FUNCTION_BLOCK FB_List_Test EXTENDS TcUnit.FB_TestSuite
VAR
END_VAR

THIS^.Size_And_Is_Empty();
THIS^.Append_And_Get();
THIS^.Prepend_And_Get();
THIS^.Append_And_Reverse();
THIS^.Append_Find_And_Get();
THIS^.Remove_Tests();
THIS^.Set_And_Get();

// Test appending multiple elements and verify their order and values using the get method.
METHOD Append_And_Get
VAR_INST
	fbList 		: FB_List;
	
	arbValue 	: ARRAY[0..2] OF BOOL := [TRUE, TRUE];
	arnValue 	: ARRAY[0..2] OF INT := [33, 33];
	arsValue 	: ARRAY[0..2] OF STRING := ['I love cats.', 'I love cats.'];
	arwsValue 	: ARRAY[0..2] OF WSTRING := ["I love dogs.", "I love dogs."];
	arfValue 	: ARRAY[0..2] OF LREAL := [21.3, 21.3];
END_VAR
TcUnit.TEST('Append_And_Get');

	fbList
		.Append(arbValue[0])
		.Append(arnValue[0])
		.Append(arsValue[0])
		.Append(arwsValue[0])
		.Append(arfValue[0]);
		
	fbList
		.Get(0, arbValue[2])
		.Get(1, arnValue[2])
		.Get(2, arsValue[2])
		.Get(3, arwsValue[2])
		.Get(4, arfValue[2]);
		
	THIS^.AssertEquals_DINT(5, fbList._Count, 'List item count must be 5 after after appending items to list.');
	THIS^.AssertEquals_BOOL(arbValue[1], arbValue[2], 'Appended BOOL item is not what is expected after the get operation.');
	THIS^.AssertEquals_INT(arnValue[1], arnValue[2], 'Appended INT item is not what is expected after the get operation.');
	THIS^.AssertEquals_STRING(arsValue[1], arsValue[2], 'Appended STRING item is not what is expected after the get operation.');
	THIS^.AssertEquals_WSTRING(arwsValue[1], arwsValue[2], 'Appended STRING item is not what is expected after the get operation.');
	THIS^.AssertEquals_LREAL(arfValue[1], arfValue[2],0.01, 'Appended LREAL item is not what is expected after the get operation.');

	TEST_FINISHED();
END_METHOD

// Test appending multiple elements, reversing their order and verifiying their order and values using the get method.
METHOD Append_And_Reverse
VAR_INST
	fbList 		: FB_List;
	
	arbValue 	: ARRAY[0..2] OF BOOL := [TRUE, TRUE];
	arnValue 	: ARRAY[0..2] OF INT := [33, 33];
	arsValue 	: ARRAY[0..2] OF STRING := ['I love cats.', 'I love cats.'];
	arwsValue 	: ARRAY[0..2] OF WSTRING := ["I love dogs.", "I love dogs."];
	arfValue 	: ARRAY[0..2] OF LREAL := [21.3, 21.3];
END_VAR
TcUnit.TEST('Append_And_Reverse');

	fbList
		.Append(arbValue[0])
		.Append(arnValue[0])
		.Append(arsValue[0])
		.Append(arwsValue[0])
		.Append(arfValue[0])
		.Reverse();
		
	fbList
		.Get(4, arbValue[2])
		.Get(3, arnValue[2])
		.Get(2, arsValue[2])
		.Get(1, arwsValue[2])
		.Get(0, arfValue[2]);
		
	THIS^.AssertEquals_DINT(5, fbList._Count, 'List item count must be 5 after after appending items to list.');
	THIS^.AssertEquals_BOOL(arbValue[1], arbValue[2], 'Appended BOOL item is not what is expected after the get operation.');
	THIS^.AssertEquals_INT(arnValue[1], arnValue[2], 'Appended INT item is not what is expected after the get operation.');
	THIS^.AssertEquals_STRING(arsValue[1], arsValue[2], 'Appended STRING item is not what is expected after the get operation.');
	THIS^.AssertEquals_WSTRING(arwsValue[1], arwsValue[2], 'Appended STRING item is not what is expected after the get operation.');
	THIS^.AssertEquals_LREAL(arfValue[1], arfValue[2],0.01, 'Appended LREAL item is not what is expected after the get operation.');

	TEST_FINISHED();
END_METHOD

// Test appending multiple elements, finds them and verify values using the get method.
METHOD Append_Find_And_Get
VAR_INST
	fbList 		: FB_List;
	Idx 		: ARRAY[0..4] OF T_Position;
	arbValue 	: ARRAY[0..2] OF BOOL := [TRUE, TRUE];
	arnValue 	: ARRAY[0..2] OF INT := [33, 33];
	arsValue 	: ARRAY[0..2] OF STRING := ['I love cats.', 'I love cats.'];
	arwsValue 	: ARRAY[0..2] OF WSTRING := ["I love dogs.", "I love dogs."];
	arfValue 	: ARRAY[0..2] OF LREAL := [21.3, 21.3];
END_VAR
TcUnit.TEST('Append_Find_And_Get');

	fbList
		.Append(arbValue[0])
		.Append(arnValue[0])
		.Append(arsValue[0])
		.Append(arwsValue[0])
		.Append(arfValue[0]);

	// Make the strings dirty. 	
	arsValue[0] 	:= 'kjhsadkfjvhbkjhdfbkvsjhbfkvjhsbkfv';
	arwsValue[0] 	:= "kjhsadkfjvhbkjhdfbkvsjhbfkvjhsbkfv";
	arsValue[0] 	:= 'I love cats.';
	arwsValue[0] 	:= "I love dogs.";
		
	fbList
		.Search(arbValue[0], Index => Idx[0])
		.Search(arnValue[0], Index => Idx[1])
		.Search(arsValue[0], Index => Idx[2])
		.Search(arwsValue[0],Index => Idx[3])
		.Search(arfValue[0], Index => Idx[4]);
		
	fbList
		.Get(Idx[0], arbValue[2])
		.Get(Idx[1], arnValue[2])
		.Get(Idx[2], arsValue[2])
		.Get(Idx[3], arwsValue[2])
		.Get(Idx[4], arfValue[2]);
		
	THIS^.AssertEquals_DINT(5, fbList._Count, 'List item count must be 5 after after appending items to list.');
	THIS^.AssertEquals_BOOL(arbValue[1], arbValue[2], 'Appended BOOL item is not what is expected after the get operation.');
	THIS^.AssertEquals_INT(arnValue[1], arnValue[2], 'Appended INT item is not what is expected after the get operation.');
	THIS^.AssertEquals_STRING(arsValue[1], arsValue[2], 'Appended STRING item is not what is expected after the get operation.');
	THIS^.AssertEquals_WSTRING(arwsValue[1], arwsValue[2], 'Appended STRING item is not what is expected after the get operation.');
	THIS^.AssertEquals_LREAL(arfValue[1], arfValue[2],0.01, 'Appended LREAL item is not what is expected after the get operation.');

	TEST_FINISHED();
END_METHOD

// Test prepending multiple elements and verify their order and values using the get method.
METHOD Prepend_And_Get
VAR_INST
	fbList 		: FB_List;
	arsPrint 	: ARRAY[0..4] OF STRING;
	arbValue 	: ARRAY[0..2] OF BOOL := [TRUE, TRUE];
	arnValue 	: ARRAY[0..2] OF INT := [33, 33];
	arsValue 	: ARRAY[0..2] OF STRING := ['I love cats.', 'I love cats.'];
	arwsValue 	: ARRAY[0..2] OF WSTRING := ["I love dogs.", "I love dogs."];
	arfValue 	: ARRAY[0..2] OF LREAL := [21.3, 21.3];
END_VAR
TcUnit.TEST('Prepend_And_Get');

	fbList
		.Prepend(arbValue[0])
		.Prepend(arnValue[0])
		.Prepend(arsValue[0])
		.Prepend(arwsValue[0])
		.Prepend(arfValue[0]);
		
	fbList
		.Get(4, arbValue[2])
		.Get(3, arnValue[2])
		.Get(2, arsValue[2])
		.Get(1, arwsValue[2])
		.Get(0, arfValue[2]);
		
	THIS^.AssertEquals_DINT(5, fbList._Count, 'List item count must be 5 after after appending items to list.');
	THIS^.AssertEquals_BOOL(arbValue[1], arbValue[2], 'Appended BOOL item is not what is expected after the get operation.');
	THIS^.AssertEquals_INT(arnValue[1], arnValue[2], 'Appended INT item is not what is expected after the get operation.');
	THIS^.AssertEquals_STRING(arsValue[1], arsValue[2], 'Appended STRING item is not what is expected after the get operation.');
	THIS^.AssertEquals_WSTRING(arwsValue[1], arwsValue[2], 'Appended STRING item is not what is expected after the get operation.');
	THIS^.AssertEquals_LREAL(arfValue[1], arfValue[2],0.01, 'Appended LREAL item is not what is expected after the get operation.');

	TEST_FINISHED();
END_METHOD

// Test appending multiple elements, removing first item, verifying the size and values.
METHOD Remove_Tests
VAR_INST
	fbList 		: FB_List;
	i 			: T_Position;
	n 			: T_Capacity;
	arbValue 	: ARRAY[0..2] OF BOOL := [TRUE, TRUE];
	arnValue 	: ARRAY[0..2] OF INT := [33, 33];
	arsValue 	: ARRAY[0..2] OF STRING := ['I love cats.', 'I love cats.'];
	arwsValue 	: ARRAY[0..2] OF WSTRING := ["I love dogs.", "I love dogs."];
	arfValue 	: ARRAY[0..2] OF LREAL := [21.3, 21.3];
END_VAR
TcUnit.TEST('Remove_Tests');

	fbList
		.Append(arbValue[0])
		.Append(arnValue[0])
		.Append(arsValue[0])
		.Append(arwsValue[0])
		.Append(arfValue[0]);
		
	fbList
		.Remove(arbValue[0])
		.Get(0, arnValue[2]);
		
	THIS^.AssertEquals_DINT(4, fbList._Count, 'List item count must be 4 after appending and removing fisrt item at from the list.');
	THIS^.AssertEquals_INT(arnValue[1], arnValue[2],'');
	
	fbList
		.Prepend(arbValue[0])
		.Remove_At(2)
		.Get(2, arwsValue[2]);
		
	THIS^.AssertEquals_DINT(4, fbList._Count, 'List item count must be 4 after prepending removed item and removing item in index 2 of the list.');
	THIS^.AssertEquals_WSTRING(arwsValue[1], arwsValue[2], '');
	
	fbList
		.Insert(2, arsValue[0])
		.Remove_At(fbList._Count - 1)
		.Get(3, arwsValue[2]);
		
	THIS^.AssertEquals_DINT(4, fbList._Count, 'List item count must be 4 after inserting removed from index 2 item and removing the last item in the list.');
	THIS^.AssertEquals_WSTRING(arwsValue[1], arwsValue[2], '');

	n := fbList._Count;
	FOR i := 0 TO n DO
		fbList.Remove_At(fbList._Count - 1);
		END_FOR
		
	THIS^.AssertEquals_DINT(0, fbList._Count, 'List item count must be zero after removing all items from the back.');
	THIS^.AssertEquals_BOOL(TRUE, fbList._Is_Empty, 'List Is_Empty property must be zero TRUE removing all items from the back.');

	FOR i := 0 TO 4 DO fbList.Prepend(arwsValue); END_FOR
	
	THIS^.AssertEquals_DINT(5, fbList._Count, 'Failed to prepend items to list for checking removing all items from the front.');
	
	n := fbList._Count;
	FOR i := 0 TO n - 1 DO
		fbList.Remove_At(0);
		END_FOR
		
	THIS^.AssertEquals_DINT(0, fbList._Count, 'List item count must be zero after removing all items from the front.');
	THIS^.AssertEquals_BOOL(TRUE, fbList._Is_Empty, 'List Is_Empty property must be zero TRUE removing all items from the front.');

	TEST_FINISHED();
END_METHOD

// Test appending multiple elements and verify their order and values using the get method.
METHOD Set_And_Get
VAR_INST
	fbList 		: FB_List;
	
	arbValue 	: ARRAY[0..2] OF BOOL := [TRUE, TRUE];
	arnValue 	: ARRAY[0..2] OF INT := [33, 33];
	arsValue 	: ARRAY[0..2] OF STRING := ['I love cats.', 'I love cats.'];
	arwsValue 	: ARRAY[0..2] OF WSTRING := ["I love dogs.", "I love dogs."];
	arfValue 	: ARRAY[0..2] OF LREAL := [21.3, 21.3];
END_VAR
TcUnit.TEST('Set_And_Get');

	fbList
		.Resize(5)
		.Set(0, arbValue[0])
		.Set(1, arnValue[0])
		.Set(2, arsValue[0])
		.Set(3, arwsValue[0])
		.Set(4, arfValue[0]);
		
	fbList
		.Get(0, arbValue[2])
		.Get(1, arnValue[2])
		.Get(2, arsValue[2])
		.Get(3, arwsValue[2])
		.Get(4, arfValue[2]);
		
	THIS^.AssertEquals_DINT(5, fbList._Count, 'List item count must be 5 after after appending items to list.');
	THIS^.AssertEquals_BOOL(arbValue[1], arbValue[2], 'Get BOOL item is not what is expected after the get operation.');
	THIS^.AssertEquals_INT(arnValue[1], arnValue[2], 'Get INT item is not what is expected after the get operation.');
	THIS^.AssertEquals_STRING(arsValue[1], arsValue[2], 'Get STRING item is not what is expected after the get operation.');
	THIS^.AssertEquals_WSTRING(arwsValue[1], arwsValue[2], 'Get STRING item is not what is expected after the get operation.');
	THIS^.AssertEquals_LREAL(arfValue[1], arfValue[2],0.01, 'Get LREAL item is not what is expected after the get operation.');

	TEST_FINISHED();
END_METHOD

// 1) Test that a newly created FB_Array_List has an item count of 0 and is empty.
// 2) Test that after appending elements, the size increases accordingly and is no longer empty.
// 3) Test that after removing all elements, the size becomes 0 again and the list is empty.
METHOD Size_And_Is_Empty
VAR_INST
	fbList : FB_List;
	nValue : INT := 33;
	sValue : STRING := 'I love cats.';
END_VAR
TcUnit.TEST('Size_And_Is_Empty');

	THIS^.AssertEquals_DINT(0, fbList._Count, 'List item count must be 0.');
	THIS^.AssertEquals_BOOL(TRUE, fbList._Is_Empty, 'Is_Empty property didnt return TRUE.');
	
	fbList
		.Append(nValue)
		.Append(sValue);
	
	THIS^.AssertEquals_DINT(2, fbList._Count, 'List item count must be 2 after appending values.');
	THIS^.AssertEquals_BOOL(FALSE, fbList._Is_Empty, 'Is_Empty property didnt return FALSE after appending value.');
	
	fbList.Clear();
	
	THIS^.AssertEquals_DINT(0, fbList._Count, 'List item count must be 0 after clearing list.');
	THIS^.AssertEquals_BOOL(TRUE, fbList._Is_Empty, 'Is_Empty property didnt return TRUE after clearing list.');
	
	TEST_FINISHED();
END_METHOD

END_FUNCTION_BLOCK

(* stored: Version 1.1.0.1, ProductVersion 3.1.4024.4
   POU FB_List_Test: Id {050c675a-d104-46d6-aa32-81ab9daf327d}, SpecialFunc None
   Method Append_And_Get: Id {535304e9-c034-4b19-9b66-933654617e91}
   Method Append_And_Reverse: Id {483f3757-3f56-41f4-b18b-bdb9d1ec2949}
   Method Append_Find_And_Get: Id {d2cf8329-d126-49e6-be8c-979349ad3a66}
   Method Prepend_And_Get: Id {bc0efed3-fbba-48dc-b3e8-6228c060fc92}
   Method Remove_Tests: Id {60ff91a6-9a36-4dc9-8548-47be6da425d5}
   Method Set_And_Get: Id {562f1aa5-f7e6-460b-88ab-27dadda3d322}
   Method Size_And_Is_Empty: Id {5e2ad20f-59dc-4dff-ada1-18ed97709948} *)
